// TIA Portal V21 export
FUNCTION_BLOCK "BoxParts"   // FB42, LAD
BEGIN

REGION Network 1: TON
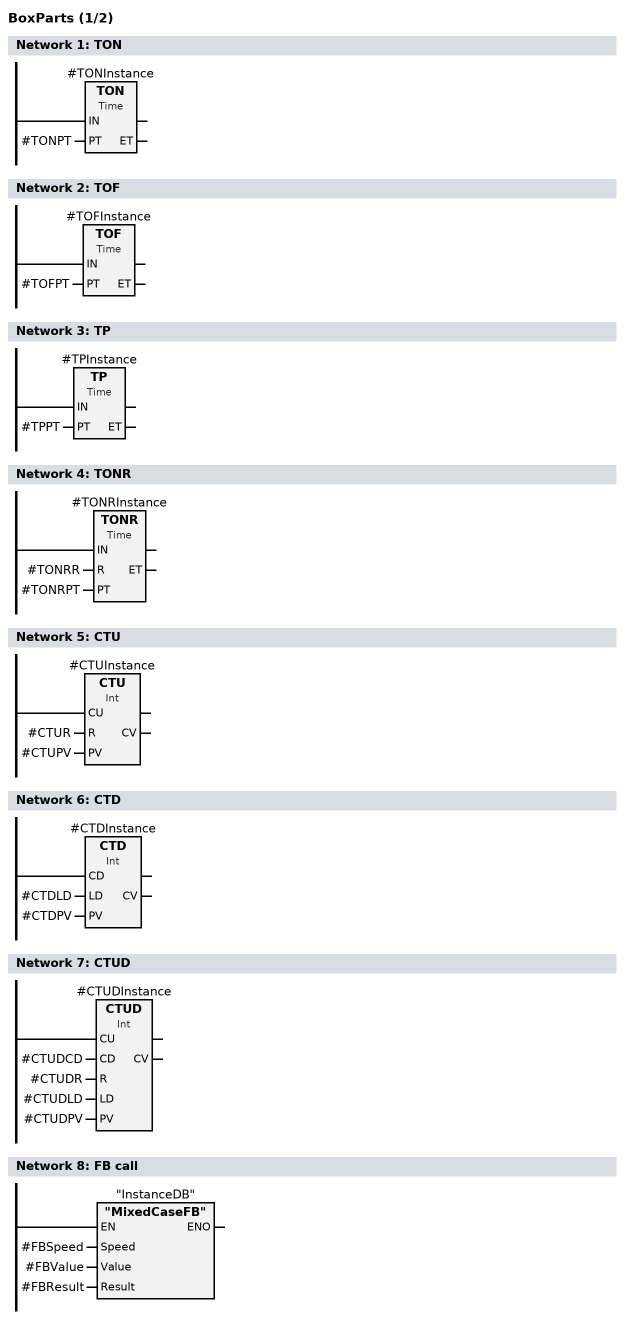
   #TONInstance.TON(IN := TRUE, PT := #TONPT);
END_REGION

REGION Network 2: TOF
   #TOFInstance.TOF(IN := TRUE, PT := #TOFPT);
END_REGION

REGION Network 3: TP
   #TPInstance.TP(IN := TRUE, PT := #TPPT);
END_REGION

REGION Network 4: TONR
   #TONRInstance.TONR(IN := TRUE, R := #TONRR, PT := #TONRPT);
END_REGION

REGION Network 5: CTU
   #CTUInstance.CTU(CU := TRUE, R := #CTUR, PV := #CTUPV);
END_REGION

REGION Network 6: CTD
   #CTDInstance.CTD(CD := TRUE, LD := #CTDLD, PV := #CTDPV);
END_REGION

REGION Network 7: CTUD
   #CTUDInstance.CTUD(CU := TRUE, CD := #CTUDCD, R := #CTUDR, LD := #CTUDLD, PV := #CTUDPV);
END_REGION

REGION Network 8: FB call
   RUNG wire#powerrail
      "InstanceDB"(Speed := #FBSpeed, Value := #FBValue, Result := #FBResult)
   END_RUNG
   // the same network as SCL:
   "InstanceDB"(Speed := #FBSpeed, Value := #FBValue, Result := #FBResult);   // "MixedCaseFB"
END_REGION

REGION Network 9: FC call
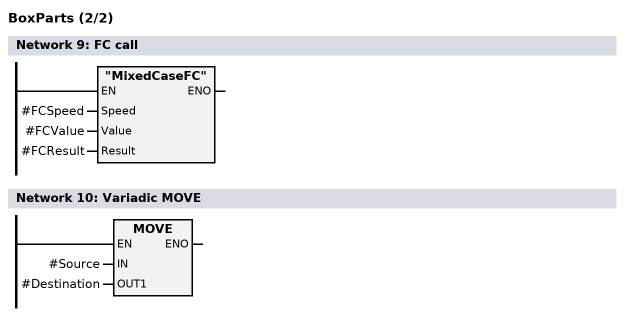
   RUNG wire#powerrail
      "MixedCaseFC"(Speed := #FCSpeed, Value := #FCValue, Result := #FCResult)
   END_RUNG
   // the same network as SCL:
   "MixedCaseFC"(Speed := #FCSpeed, Value := #FCValue, Result := #FCResult);
END_REGION

REGION Network 10: Variadic MOVE
   RUNG wire#powerrail
      { S7_GenerateENO := "TRUE" } Move(in := #Source, out1 := #Destination)
   END_RUNG
   // the same network as SCL:
   <??.?> := #Source;
END_REGION

REGION Network 11 (FBD): Word logic
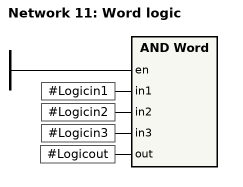
   <??.?> := #Logicin1 AND #Logicin2 AND #Logicin3 AND #Logicout;
END_REGION

REGION Network 12: Unknown fallback
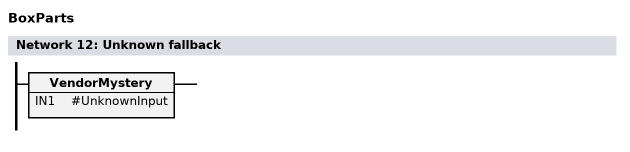
   // no SCL statement known for VendorMystery: written as a call
END_REGION
END_FUNCTION_BLOCK
